{attribute 'linkalways'} 
{attribute 'no_explicit_call' := 'This FB is a CLASS and must be accessed using methods or properties'}
{attribute 'enable_dynamic_creation'}
FUNCTION_BLOCK _ETcVnEdgeDetectionAlgorithm EXTENDS EnumDatatypeBase
VAR
	localData : ETcVnEdgeDetectionAlgorithm;
	activeData : REFERENCE TO ETcVnEdgeDetectionAlgorithm;
	enumBaseDatatype : _DINT(localData);
END_VAR

METHOD PRIVATE AddLocalEnumeration
VAR_INPUT
	Enumeration : T_MAXSTRING;
	Value : ETcVnEdgeDetectionAlgorithm;
END_VAR
AddEnumeration(Enumeration, Value);
END_METHOD

PROPERTY PUBLIC Address : PVOID
GET
Address := ADR(activeData);
END_GET
END_PROPERTY

METHOD PUBLIC ClearReference
VAR_INPUT
END_VAR
activeData REF= localData;
SetBaseDatatypeReference();
END_METHOD

METHOD PUBLIC Clone : I_Datatype
VAR
    pClone : POINTER TO _ETcVnEdgeDetectionAlgorithm;
END_VAR
pClone := __NEW(_ETcVnEdgeDetectionAlgorithm(InitialValue := Value));
Clone := pClone^;
END_METHOD

METHOD FB_init : BOOL
VAR_INPUT
	bInitRetains : BOOL; // if TRUE, the retain variables are initialized (warm start / cold start)
	bInCopyCode : BOOL;  // if TRUE, the instance afterwards gets moved into the copy code (online change)
	InitialValue : ETcVnEdgeDetectionAlgorithm;
END_VAR
localData := InitialValue;
AddBaseDatatype(enumBaseDatatype);
ClearReference();

AddLocalEnumeration('TCVN_EDA_INTERPOLATION', ETcVnEdgeDetectionAlgorithm.TCVN_EDA_INTERPOLATION);
AddLocalEnumeration('TCVN_EDA_APPROX_ERF', ETcVnEdgeDetectionAlgorithm.TCVN_EDA_APPROX_ERF);
AddLocalEnumeration('TCVN_EDA_APPROX_GAUSSIAN', ETcVnEdgeDetectionAlgorithm.TCVN_EDA_APPROX_GAUSSIAN);
END_METHOD

PROPERTY PUBLIC Identifier : T_MAXSTRING
GET
Identifier := 'ETcVnEdgeDetectionAlgorithm';
END_GET
END_PROPERTY

METHOD IsEnumeratorValueEqual : BOOL
VAR_INPUT
	Enumerator : I_KeyValueForwardEnumerator;
END_VAR
VAR
	storedValue : ETcVnEdgeDetectionAlgorithm;
END_VAR
IF NOT Enumerator.TryGet(storedValue) THEN
	RETURN;
END_IF

IsEnumeratorValueEqual := storedValue = activeData;
END_METHOD

METHOD PUBLIC MakeReferenceTo
VAR_INPUT
	ReferenceTarget : REFERENCE TO ETcVnEdgeDetectionAlgorithm;
END_VAR
activeData REF= ReferenceTarget;
SetBaseDatatypeReference();
END_METHOD

METHOD PROTECTED SetBaseDatatypeReference
VAR_INPUT
END_VAR
enumBaseDatatype.MakeReferenceTo(activeData);
END_METHOD

PROPERTY PUBLIC Size : UDINT
GET
Size := SIZEOF(activeData);
END_GET
END_PROPERTY

METHOD TryMakeReferenceTo : BOOL
VAR_INPUT
	Target : I_Datatype;
END_VAR
VAR
	targetAsEnum : I_EnumDatatype;
	pTargetData : POINTER TO ETcVnEdgeDetectionAlgorithm;
END_VAR
IF NOT Target.TryResolveAsEnumDatatype(targetAsEnum) THEN
	RETURN;
END_IF

IF targetAsEnum.Identifier <> Identifier THEN
	RETURN;
END_IF

pTargetData := Target.Address;
activeData REF= pTargetData^;
SetBaseDatatypeReference();
TryMakeReferenceTo := TRUE;
END_METHOD

PROPERTY PUBLIC Value : ETcVnEdgeDetectionAlgorithm
GET
Value := activeData;
END_GET
SET
activeData := Value;
END_SET
END_PROPERTY

END_FUNCTION_BLOCK

(* stored: Version 1.1.0.1, ProductVersion 3.1.4024.12
   POU _ETcVnEdgeDetectionAlgorithm: Id {de3327d9-628b-0db8-070f-b6ec3e9cfed8}, SpecialFunc None
   Folder Constructor: Id {163cf6a0-f511-071e-20fa-813a2df9bf96}
   Folder Private: Id {fa96855c-e46a-09e8-18d9-cd7d699408c7}
   Folder Protected: Id {81f72d85-df5c-0d10-25bf-c5676d71d58f}
   Method AddLocalEnumeration: Id {c7807dc8-fcd2-0167-2c69-db3e14617561}
   Property Address: Id {fd1129ea-2683-02b4-1b4b-23165bf232e5}
   Get Get: Id {9ca24ffe-0aa1-007f-2ae9-eadabd6c358e}
   Method ClearReference: Id {e5f49816-fc55-08c6-0902-0a2a0f521659}
   Method Clone: Id {93dcc90a-ca49-0669-2de3-8775364a3c48}
   Method FB_init: Id {499c5acc-ee1f-048c-274d-37da243b2af5}
   Property Identifier: Id {73c0b194-9924-0dcf-2ac0-b517abdb4f5b}
   Get Get: Id {2391be6c-42a0-0570-0938-859bb6badf5f}
   Method IsEnumeratorValueEqual: Id {15a04b32-a76a-0a9a-0ce5-ab7589c338e2}
   Method MakeReferenceTo: Id {96185666-00ce-04b4-2ca1-41455ce3c251}
   Method SetBaseDatatypeReference: Id {34da90ee-18ff-0fcb-0b76-51877e250af5}
   Property Size: Id {daa2e842-42b4-08e4-0c80-ad85a3209b54}
   Get Get: Id {ae48c7f4-1abe-0765-0683-2aa5f595fb2c}
   Method TryMakeReferenceTo: Id {7b1ff354-ecf7-0aaf-01ca-730cbb69bce2}
   Property Value: Id {961ce8f3-bf3e-0537-187a-30ab8e162096}
   Get Get: Id {bb0abdb4-7053-07e8-3dd2-c591c18a5e7c}
   Set Set: Id {08eee3c9-39d1-055b-191e-944ae51f1070} *)
